PROGRAM MAIN
VAR
END_VAR

END_PROGRAM

(* stored: Version 1.1.0.1
   POU MAIN: Id {a4dcdf13-c3d7-4037-8603-447a8fa6602f} *)
